TYPE ST_SettingsDoorLock :
STRUCT
	tUnlockingRequestTimeout : TIME := T#30S; //Unlocking request timeout [default: 30s]
	bAutoLockAtInit : BOOL := TRUE; //Automatically lock at init (if door is closed) [Y/N]
END_STRUCT
END_TYPE

(* stored: Version 1.1.0.1, ProductVersion 3.1.4024.12
   DUT ST_SettingsDoorLock: Id {959adbfb-3b17-44ae-9aa1-564241597ba9} *)
